INTERFACE ITF_BaseControlElement EXTENDS ITF_BaseComponent

(*			
	EVERDE sp. z o.o.
	Rafał Osajda		31.03.2025		TC 4024.66
	Flaga że w tej sesji pracy maszyny element został już wybazowany
*)
METHOD PUBLIC HomingGetDone : BOOL
VAR_INPUT
END_VAR
END_METHOD

(*			
	EVERDE sp. z o.o.
	Rafał Osajda		11.04.2025		TC 4024.66
	Zwraca czy bazowanie jest potrzebne
*)
METHOD PUBLIC HomingGetIsNeeded : BOOL
VAR_INPUT
END_VAR
END_METHOD

(*			
	EVERDE sp. z o.o.
	Rafał Osajda		27.05.2025		TC 4024.66
	Uruchomienie metody bazowania
*)
METHOD PUBLIC HomingStart
VAR_INPUT
END_VAR
END_METHOD

(*			
	EVERDE sp. z o.o.
	Rafał Osajda		30.04.2025		TC 4024.66
	Zwraca czy element jest czymś zajety
*)
METHOD PUBLIC IsDoNothing : BOOL
END_METHOD

(*			
	EVERDE sp. z o.o.
	Rafał Osajda		30.04.2025		TC 4024.66
	Zwraca czy element jest w pozycji 0 - referencyjnej
*)
METHOD PUBLIC IsPosition0 : BOOL
END_METHOD

METHOD PUBLIC LinkSS1 : BOOL
VAR_INPUT
	fbSS1			: ITF_BaseFlagGet;
END_VAR
END_METHOD

METHOD PUBLIC LinkSTO : BOOL
VAR_INPUT
	fbSTO			: ITF_BaseFlagGet;
END_VAR
END_METHOD

(*			
	EVERDE sp. z o.o.
	Rafał Osajda		31.03.2025		TC 4024.66
	Zwraca status zasilania	
*)
METHOD PUBLIC PowerGetStatus : BOOL
VAR_INPUT
END_VAR
END_METHOD

(*			
	EVERDE sp. z o.o.
	Rafał Osajda		31.03.2025		TC 4024.66
	Wyłączenie zasilania
*)
METHOD PUBLIC PowerTurnOff : BOOL
VAR_INPUT
END_VAR
END_METHOD

(*			
	EVERDE sp. z o.o.
	Rafał Osajda		31.03.2025		TC 4024.66
	Uruchomienie zasialania
*)
METHOD PUBLIC PowerTurnOn
VAR_INPUT
END_VAR
END_METHOD

END_INTERFACE

(* stored: Version 1.1.0.1
   Itf ITF_BaseControlElement: Id {ad3f64dc-ad28-0928-11ba-a3b4f43ec05a}
   Folder Bazowanie: Id {683853aa-b098-0b06-1f91-4b58f7657d20}
   Folder WiazanieZmiennych: Id {3ea49384-a761-0669-1c6e-519f81bf24fd}
   Folder Zasilanie: Id {5277a279-1f79-0b64-1781-5812a3c092e7}
   Method HomingGetDone: Id {fde5b151-5c08-07ea-2de6-6340c0692556}
   Method HomingGetIsNeeded: Id {af92a4dc-5ebd-0ea2-0b2f-d3ed007008d4}
   Method HomingStart: Id {4da12ea9-04a5-0fd9-182f-16900ea540df}
   Method IsDoNothing: Id {ffddb488-5890-0adf-06a6-f772df0e09cc}
   Method IsPosition0: Id {44c176d3-d246-039d-2b7a-13136bdef39e}
   Method LinkSS1: Id {db097555-ff7f-040e-3bc7-54bad7054deb}
   Method LinkSTO: Id {af004b13-a591-0136-09de-53edc6e3a981}
   Method PowerGetStatus: Id {365f79a7-e897-0e0f-0996-f98b05052eb0}
   Method PowerTurnOff: Id {c3b82c4f-b776-099b-1ee8-48f958193ea3}
   Method PowerTurnOn: Id {a4b9ee87-99e7-08e4-233a-a1dfefa8327a} *)
